PROGRAM MAIN
VAR
	bInit: BOOL;
	sStart: STRING;
END_VAR

//Develolep BY Kauê Koschitz Roratto
//https://github.com/KaueKoschitzRoratto
//https://www.linkedin.com/in/kauekoschitzroratto/
//kaue.roratto@outlook.com.br

IF bInit THEN
	sStart:= 'project Started';
END_IF

END_PROGRAM

(* stored: Version 1.1.0.1, ProductVersion 3.1.4024.9
   POU MAIN: Id {3c6388f7-e206-4478-ac30-7b1468125055}, SpecialFunc None *)
